{attribute 'linkalways'} 
{attribute 'no_explicit_call' := 'This FB is a CLASS and must be accessed using methods or properties'}
{attribute 'enable_dynamic_creation'}
FUNCTION_BLOCK Node_ContainerType_Vector_TcVnVector4_LREAL EXTENDS Node
VAR
    out : _GUID;
END_VAR

METHOD PUBLIC  Clone : I_Node
VAR
	pNode : POINTER TO Node_ContainerType_Vector_TcVnVector4_LREAL;
END_VAR
pNode := __NEW(Node_ContainerType_Vector_TcVnVector4_LREAL);
Clone := pNode^;
END_METHOD

METHOD FB_init : BOOL
VAR_INPUT
	bInitRetains : BOOL; // if TRUE, the retain variables are initialized (warm start / cold start)
	bInCopyCode : BOOL;  // if TRUE, the instance afterwards gets moved into the copy code (online change)
END_VAR
AddOutput('out', out);
END_METHOD

METHOD PROTECTED OnExecute
out.Value := ContainerType_Vector_TcVnVector4_LREAL;
END_METHOD

END_FUNCTION_BLOCK

(* stored: Version 1.1.0.1, ProductVersion 3.1.4026.17
   POU Node_ContainerType_Vector_TcVnVector4_LREAL: Id {e8191bb8-f70f-0557-0714-657b6968f957}, SpecialFunc None
   Folder Constructor: Id {afc13c23-8c6f-0ee5-0667-00212cdeae04}
   Method Clone: Id {9d9fd5e8-50fb-0e72-3dd1-618a9605cb17}
   Method FB_init: Id {8fc3b468-f72a-0a7b-2ce2-1cec95baee2b}
   Method OnExecute: Id {c3c8c663-8a79-0847-3e7e-0aab2e85d96b} *)
